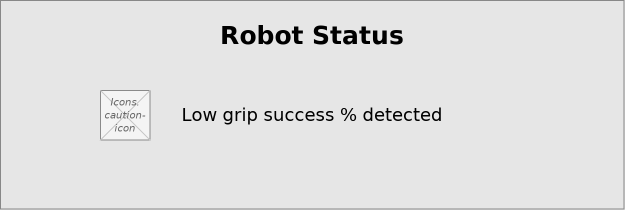
VISUALIZATION RobotStatusPopup  // 625x210
    Textfield (212,10 200x50), "Robot Status"
    Image (100,90 50x50), image: Icons.caution-icon
    Textfield (162,100 300x30), "Low grip success % detected"
END_VISUALIZATION

(* stored: Version 1.1.0.1, ProductVersion 3.1.4024.15
   Visu RobotStatusPopup: Id {988c55d3-033e-48ee-b85c-5c5d77411dc5} *)
